TYPE ST_ModePermits :
STRUCT
    bAllowMotion : BOOL;
    bAllowJog : BOOL;
    bAllowHoming : BOOL;
    bAllowAutoStart : BOOL;
    bAllowModeChange : BOOL;
    bAllowConfigEdit : BOOL;
    bAllowAlarmReset : BOOL;
END_STRUCT
END_TYPE

(* stored: Version 1.1.0.1
   DUT ST_ModePermits: Id {70DCFFFD-4D05-8CF3-2969-A9C111B04EC6} *)
